TEXTLIST TextList_VVAT_3P
  0 = 'ouv' | FR: 'Ouvrir' | EN: 'Open'
  1 = 'ferme' | FR: 'Fermer' | EN: 'Close'
  2 = 'lam' | FR: 'Laminer' | EN: 'Throttle'
   = ''
END_TEXTLIST

(* stored: Version 1.1.0.1, ProductVersion 3.1.4024.10
   TextList TextList_VVAT_3P: Id {3993eac9-3129-48c2-b2eb-d4dd775e723e} *)
